RoboDK station: RobodkBasico-2.rdk

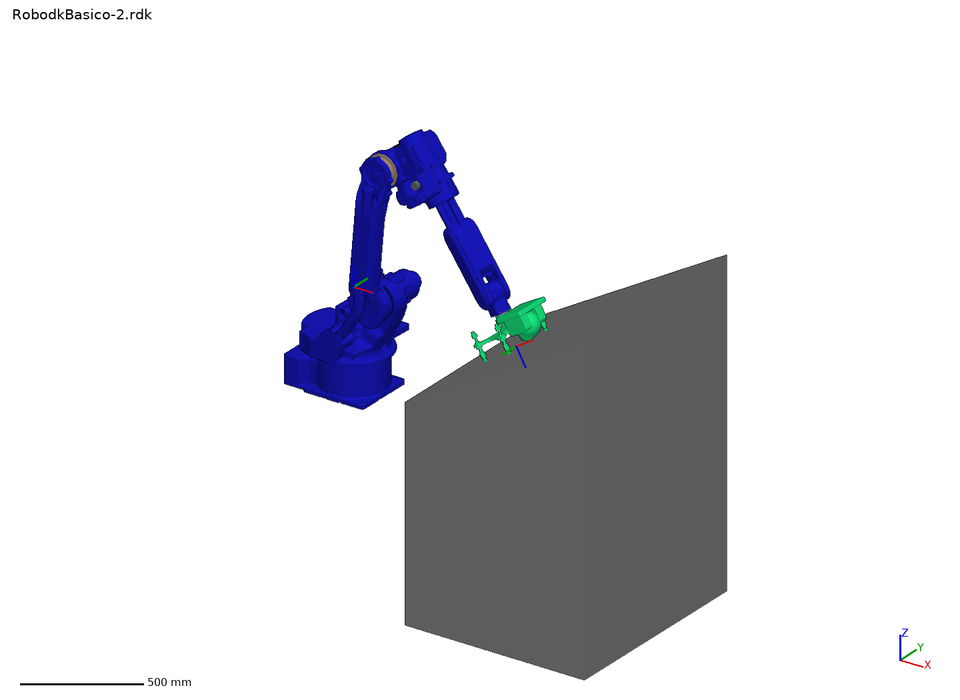
[picture v0: the station drawn from its stored meshes, robots at their saved joint values, targets as dots, program paths as lines]
Station Robodk (2) (saved by RoboDK 5.9.1). Poses are relative to the parent item; angles as X-Y-Z fixed-axis rotations.
  - frame Motoman MH6 Base at (0, 0, 450) mm
    - robot Motoman MH6: 6 axes, payload 6 kg, reach 1422 mm, repeatability 0.08 mm, weight 130 kg
        modified DH rows (alpha deg, a mm, theta deg, d mm): 0, 0, 0, 450; -90, 152, -90, 0; 0, 614, 0, 0; -90, 155, 0, 640; 90, 0, 90, 0; -90, 0, 0, 95
        base shift (0, 0, -450) mm
        joint limits [-170, -90, -175, -180, -45, -360] to [170, 155, 250, 180, 225, 360]; home [0, 0, 0, 0, 0, 0]; saved at [-2.798, 5.147, -49.137, -13.706, 84.087, 16.059]
      - tool Ventosas, TCP at (0, 0, 190) mm, size 250 x 290 x 148 mm
    - frame Frame_from_Target1 at (823.2, -34.49, -21.13) mm, rotated rx -180 ry -30 rz 0 deg
  - object CAJA2 at (1600, 500, 300) mm, rotated rx 180 ry 0 rz 0 deg, size 886.4 x 1000 x 1511.7 mm, geometry from CAJA2.stp
  - Python program RosPolar (listed below)

--- Python program RosPolar ---
from robodk.robolink import *    # API para comunicarte con RoboDK
from robodk.robomath import *    # Funciones matemáticas
import math

#------------------------------------------------
# 1) Conexión a RoboDK e inicialización
#------------------------------------------------
RDK = Robolink()
# Elegir un robot (si hay varios, aparece un popup)
robot = RDK.ItemUserPick("Selecciona un robot", ITEM_TYPE_ROBOT)
if not robot.Valid():
    raise Exception("No se ha seleccionado un robot válido.")

# Conectar al robot físico (descomentado para pruebas reales)
#if not robot.Connect():
#    raise Exception("No se pudo conectar al robot. Verifica que esté en modo remoto y que la configuración sea correcta.")
#if not robot.ConnectedState():
#    raise Exception("El robot no está conectado correctamente. Revisa la conexión.")
#print("Robot conectado correctamente.")

#------------------------------------------------
# 2) Cargar el Frame (ya existente) donde quieres dibujar
#------------------------------------------------
frame_name = "Frame_from_Target1"
frame = RDK.Item(frame_name, ITEM_TYPE_FRAME)
if not frame.Valid():
    raise Exception(f'No se encontró el Frame "{frame_name}" en la estación.')

# Asignamos este frame al robot
robot.setPoseFrame(frame)
# Usamos la herramienta activa
robot.setPoseTool(robot.PoseTool())

# Ajustes de velocidad y blending
robot.setSpeed(200)   # mm/s - Velocidad reducida para mejor precisión
robot.setRounding(3)  # blending (radio de curvatura)

#------------------------------------------------
# 3) Parámetros para las cardioides concéntricas
#------------------------------------------------
num_points = 360       # Puntos por cardioide (1 punto por grado)
num_cardioides = 5     # Número total de cardioides
z_surface = 0          # Z=0 en el plano del frame
z_safe = 50            # Altura segura para aproximarse y salir

# Offset para desplazar toda la trayectoria
offset_x = 300         # mm - Desplazamiento en X (positivo = hacia adelante)
offset_y = 100           # mm - Desplazamiento en Y (opcional)
offset_z = 0           # mm - Desplazamiento en Z (opcional)

# Radio del círculo contenedor
radio_circulo = 300    # mm - Reducido para evitar límites del robot (ajusta según tu espacio de trabajo)

# Calculamos el parámetro 'a' máximo para que la cardioide más grande
# quepa dentro del círculo. Para una cardioide r = a(1 + cos(θ)),
# el radio máximo es 2a (cuando θ = 0)
a_max = radio_circulo / 2

# Parámetros 'a' para cada cardioide (de mayor a menor)
parametros_a = []
for i in range(num_cardioides):
    # Distribuimos los tamaños uniformemente
    factor = (num_cardioides - i) / num_cardioides
    a = a_max * factor
    parametros_a.append(a)

print(f"Dibujando {num_cardioides} cardioides concéntricas")
print(f"Radio del círculo contenedor: {radio_circulo} mm")
print(f"Parámetros 'a': {[round(a, 1) for a in parametros_a]}")

#------------------------------------------------
# 4) Función para dibujar una cardioide
#------------------------------------------------
def dibujar_cardioide(robot, a, z_surface, z_safe, num_points, offset_x=0, offset_y=0, offset_z=0):
    """
    Dibuja una cardioide con parámetro 'a'
    Ecuación: r = a(1 + cos(θ))
    """
    print(f"Dibujando cardioide con a = {a:.1f} mm (offset X: {offset_x}, Y: {offset_y}, Z: {offset_z})")

    # Calcular el punto inicial (θ = 0)
    theta_inicial = 0
    r_inicial = a * (1 + math.cos(theta_inicial))
    x_inicial = r_inicial * math.cos(theta_inicial) + offset_x
    y_inicial = r_inicial * math.sin(theta_inicial) + offset_y
    z_inicial = z_surface + offset_z

    # Ir al punto inicial en altura segura
    robot.MoveJ(transl(x_inicial, y_inicial, z_inicial + z_safe))
    # Bajar a la superficie
    robot.MoveL(transl(x_inicial, y_inicial, z_inicial))

    # Dibujar la cardioide completa (0 a 2π)
    for i in range(1, num_points + 1):
        # Ángulo actual
        theta = (2 * math.pi * i) / num_points

        # Calcular radio para la cardioide: r = a(1 + cos(θ))
        r = a * (1 + math.cos(theta))

        # Convertir a coordenadas cartesianas y aplicar offset
        x = r * math.cos(theta) + offset_x
        y = r * math.sin(theta) + offset_y
        z = z_surface + offset_z

        # Mover linealmente
        robot.MoveL(transl(x, y, z))

    # Subir a altura segura al terminar
    robot.MoveL(transl(x, y, z + z_safe))

#------------------------------------------------
# 5) Dibujar todas las cardioides (de mayor a menor)
#------------------------------------------------
print("Iniciando el dibujo de las cardioides...")

for i, a in enumerate(parametros_a):
    print(f"\n--- Cardioide {i+1}/{num_cardioides} ---")
    dibujar_cardioide(robot, a, z_surface, z_safe, num_points, offset_x, offset_y, offset_z)

#------------------------------------------------
# 6) Opcional: Dibujar el círculo contenedor
#------------------------------------------------
dibujar_circulo = True  # Cambia a False si no quieres el círculo

if dibujar_circulo:
    print(f"\n--- Dibujando círculo contenedor (radio = {radio_circulo} mm) ---")

    # Punto inicial del círculo (con offset)
    x_inicial = radio_circulo + offset_x
    y_inicial = 0 + offset_y
    z_inicial = z_surface + offset_z

    # Ir al punto inicial
    robot.MoveJ(transl(x_inicial, y_inicial, z_inicial + z_safe))
    robot.MoveL(transl(x_inicial, y_inicial, z_inicial))

    # Dibujar el círculo
    puntos_circulo = 72  # 5 grados por punto
    for i in range(1, puntos_circulo + 1):
        theta = (2 * math.pi * i) / puntos_circulo
        x = radio_circulo * math.cos(theta) + offset_x
        y = radio_circulo * math.sin(theta) + offset_y
        z = z_surface + offset_z
        robot.MoveL(transl(x, y, z))

    # Subir al terminar
    robot.MoveL(transl(x, y, z + z_safe))

#------------------------------------------------
# 7) Posición final
#------------------------------------------------
# Volver al centro desplazado en altura segura
robot.MoveJ(transl(0 + offset_x, 0 + offset_y, z_surface + offset_z + z_safe))


# Primera letra J (Juan)
robot.MoveL(transl(300, -300, z_surface + z_safe))
robot.MoveL(transl(300, -300, z_surface))
robot.MoveL(transl(200, -300, z_surface))
robot.MoveC(transl(150, -350, z_surface), transl(200, -400, z_surface) )
robot.MoveJ(transl(200, -400, z_surface + z_safe))

# Segunda letra M (Miguel)
robot.MoveJ(transl(-50, -300, z_surface + z_safe))
robot.MoveL(transl(-50, -300, z_surface))
robot.MoveL(transl(100, -300, z_surface))
robot.MoveL(transl(-50, -350, z_surface))
robot.MoveL(transl(100, -400, z_surface))
robot.MoveL(transl(-50, -400, z_surface))
robot.MoveJ(transl(-50, -400, z_surface + z_safe))

# Tercera letra D (Dixon)
robot.MoveJ(transl(-250, -400, z_surface + z_safe))
robot.MoveL(transl(-250, -400, z_surface))
robot.MoveL(transl(-100, -400, z_surface))
robot.MoveL(transl(-100, -375, z_surface))
robot.MoveC(transl(-175, -300, z_surface), transl(-250, -375, z_surface))
robot.MoveL(transl(-250, -400, z_surface))
robot.MoveJ(transl(-250, -400, z_surface + z_safe))

# Movimiento al origen del Frame + z_ safe
robot.MoveJ(transl(0, 0, z_surface + z_safe))

print(f"\n¡Patrón de cardioides completado en el frame '{frame_name}'!")
print(f"Se dibujaron {num_cardioides} cardioides concéntricas dentro de un círculo de {radio_circulo} mm")
